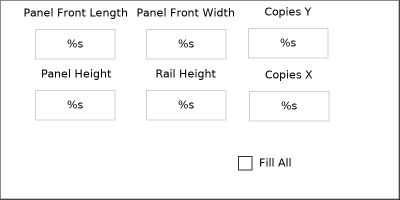
VISUALIZATION V_ProductionBorgoFlaps  // 400x200
VAR_IN_OUT
	HMI : ST_PackMLBaseModule_HMI;
	HMI_GantryXYZ : ST_GantryXYZ_HMI;
	HMI_Recipe : ST_RecipeBuilder_HMI;
END_VAR
    RoundedRectangle (0,0 400x200)
    Textfield (35,29 80x30), "%s", text variable: HMI_Recipe.Config.PanelFrontLength
        OnMouseClick: write the text variable via VisuDialogs.Numpad, min HMI_Recipe.Limits.PanelFrontLength.MinVal, max HMI_Recipe.Limits.PanelFrontLength.MaxVal
    Label (18,3 116x20), "Panel Front Length"
    Textfield (146,29 80x30), "%s", text variable: HMI_Recipe.Config.PanelFrontWidth
        OnMouseClick: write the text variable via VisuDialogs.Numpad, min HMI_Recipe.Limits.PanelFrontWidth.MinVal, max HMI_Recipe.Limits.PanelFrontWidth.MaxVal
    Label (97,3 178x20), "Panel Front Width"
    Textfield (35,90 80x30), "%s", text variable: HMI_Recipe.Config.PanelHeight
        OnMouseClick: write the text variable via VisuDialogs.Numpad, min HMI_Recipe.Limits.PanelHeight.MinVal, max HMI_Recipe.Limits.PanelHeight.MaxVal
    Label (19,64 115x20), "Panel Height"
    Textfield (146,90 80x30), "%s", text variable: HMI_Recipe.Config.RailHeightCorrection
        OnMouseClick: write the text variable via VisuDialogs.Numpad, min HMI_Recipe.Limits.RailHeightCorrection.MinVal, max HMI_Recipe.Limits.RailHeightCorrection.MaxVal
    Label (135,64 102x20), "Rail Height"
    Checkbox (236,148 72x30), "Fill All", variable: HMI_Recipe.Config.FillAll
    Textfield (249,91 80x30), "%s", text variable: HMI_Recipe.Config.RequestedCopiesX, input disabled if: MAIN.Seedra.RecipeConfig_HMI.Config.FillAll
        OnMouseClick: write the text variable via VisuDialogs.Numpad, min 1, max MAIN.Seedra.RecipeConfig_HMI.Limits.RequestedCopiesX.MaxVal
    Label (238,65 102x20), "Copies X"
    Textfield (248,28 80x30), "%s", text variable: HMI_Recipe.Config.RequestedCopiesY, input disabled if: MAIN.Seedra.RecipeConfig_HMI.Config.FillAll
        OnMouseClick: write the text variable via VisuDialogs.Numpad, min 1, max MAIN.Seedra.RecipeConfig_HMI.Limits.RequestedCopiesY.MaxVal
    Label (237,2 102x20), "Copies Y"
END_VISUALIZATION

(* stored: Version 1.1.0.1, ProductVersion 3.1.4024.15
   Visu V_ProductionBorgoFlaps: Id {571e1921-2ea2-4d68-a038-db63e03e77f7} *)
